PROGRAM POU
VAR
END_VAR

GVL_1.bYAwVar1:=true;

END_PROGRAM

(* stored: Version 1.1.0.1, ProductVersion 3.1.4022.17
   POU POU: Id {84837b54-8a87-4787-98ed-252eb95b0351}, SpecialFunc None *)
